Fanuc KAREL source: kt00933.KL

PROGRAM KT00933
%NOLOCKGROUP
VAR
ENTRY:INTEGER;PNAME : STRING[80];VNAME : STRING[80];STATUS:INTEGER;VALUE:INTEGER
BEGIN
--
--
--
--
ENTRY=0
PNAME=''
VNAME='VALUE'
GET_VAR(ENTRY,PNAME,VNAME,VALUE,STATUS)
END KT00933
